(* IEC 61131-3 sources: ml2plc/benchmarks/st (part 4) *)

(* ---- GRU2_straton.st ---- *)
FUNCTION_BLOCK GRU2_FB

    (* Model Inputs/Outputs *)
VAR_INPUT
    input_data : REAL;
END_VAR

VAR_OUTPUT
    output_data : ARRAY[0..2] OF REAL;
END_VAR

VAR
    CONSTANT weights_0_u : ARRAY[0..35] OF REAL := [-1.26034391, 0.836788237, -0.74071312, -1.66741002, -1.1549176, -1.52132487, -1.16551328, -1.43403518, -1.60023963, -1.46855605, -1.58754134, -1.517748, -1.31009662, -0.703322828, -1.11610091, 0.108651124, -1.24668264, -1.7667824, -1.78982019, -1.47540379, -1.49926209, -1.13290668, -1.73071063, -1.48351586, -1.53246319, -2.03121448, -1.50697207, -1.17749131, -1.91584527, -1.08492792, -0.994556248, -1.55253255, -1.03130341, -1.2640295, -0.178557396, -1.63782966];
    CONSTANT recurrent_0_u : ARRAY[0..1295] OF REAL := [-0.0342628956, 0.033126276, 0.0130427806, 0.0238829348, -0.0667412207, -0.0413707495, -0.0313988812, 0.0143869575, 0.190381631, -0.0726102442, 0.0838638023, 0.0527294315, -0.0637015849, -0.182236433, 0.144636199, -0.122772858, -0.141192406, -0.00673655141, 0.0763217956, -0.0320057683, 0.0996292979, -0.137748078, -0.0618084669, -0.0315994285, -0.062908709, -0.00729163829, -0.0906494558, -0.137917697, -0.0289651398, 0.0414582938, -0.0709736273, -0.0059862812, 0.0197576638, -0.0750913471, -0.142621666, -0.0388273448, -0.260161608, 0.00932510011, 0.00876244251, -0.12344873, -0.0972604752, -0.0141034368, 0.07111267, 0.00913770497, 0.170134529, 0.0203112364, -0.0925216526, -0.0673360229, -0.0160743687, 0.117756821, 0.134309813, -0.0970909521, 0.0523982346, -0.0415440686, -0.0711917579, 0.0170196127, -0.045774959, -0.0370751619, -0.0704077557, 0.0188004524, -0.0777330324, 0.283721894, -0.16303502, 0.0651905835, 0.0264630243, 0.0179281905, -0.138563886, 0.0722385198, -0.0791174024, -0.0230214931, -0.163337797, -0.0849895626, 0.00793311652, 0.00964403804, -0.0900170207, -0.0211868752, 0.065747194, 0.141165093, 0.0130933337, -0.126985207, 0.0847581699, -0.195722729, -0.0474834777, -0.0756620616, 0.0745357648, 0.11035046, 0.0613997541, 0.0489263199, 0.0219242349, 0.0518789999, 0.180661157, -0.141433775, -0.0488601774, 0.0343847387, 0.0521875918, -0.0937664136, -0.0139141269, 1.37788593e-05, -0.0523182154, -0.0222289097, 0.199464455, -0.195190653, -0.0105472393, 0.0335475393, 0.17911391, 0.032945402, 0.0335034542, 0.146120399, -0.0346618779, -0.027050646, -0.0628796816, -0.126079142, -0.0608317778, -0.144880667, -0.170438543, -0.139052421, 0.0964757726, -0.0888345987, 0.140413404, -0.00511395978, -0.169440314, -0.0679477602, 0.179598868, 0.0536571033, -0.100946359, 0.297387779, 0.14612335, -0.0515739471, -0.0920707807, 0.1155788, 0.122627199, 0.173509136, -0.0269757025, 0.0626975074, 0.0153822703, -0.128492385, -0.193825796, 0.0969658792, 0.0116878124, 0.0272942241, 0.0452310033, 0.00160261057, 0.264178902, -0.103370436, 0.0297610722, -0.0913388878, -0.0183291547, 0.0166632738, 0.119481407, -0.0304607637, -0.0763635635, -0.000451272033, -0.107587576, -0.151274115, 0.122772105, -0.031456992, -0.000585220521, -0.00406094966, -0.139671892, 0.0299809463, -0.102254301, 0.0713162273, 0.00914381258, -0.0205416568, -0.0607767105, 0.0461449251, -0.0858086646, -0.0383039862, -0.0823218748, 0.0483131632, 0.0267805085, 0.193337917, 0.163598657, 0.0458281264, -0.0303147305, -0.19125393, -0.0151128527, 0.00750773214, 0.0093731042, -0.132128522, -0.0926906914, 0.0911830217, -0.127907664, 0.0237907302, 0.00307789678, 0.0957302004, 0.11556039, 0.172038779, 0.0433095135, -0.0654063001, 0.0514559746, -0.00690185279, 0.0779523849, -0.05985808, -0.135543838, 0.0494517833, 0.0334763303, 0.0388004482, -0.172183558, -0.113222495, -0.142196029, 0.139659673, -0.10881792, 0.0211461224, -0.0613673106, 0.125337034, 0.052437298, 0.0480097719, 0.0614684746, -0.0621075481, 0.215367347, 0.137130678, -0.0973720923, 0.0115704983, 0.254007638, -0.106283039, 0.165332898, 0.173523873, -0.0684746727, 0.0595950186, -0.0305053927, -0.0180566646, 0.0267004631, -0.0547558889, 0.207268775, 0.0180881377, 0.153428495, 0.0346085951, 0.00634628395, -0.0340505242, 0.0254321843, -0.0179827698, -0.110346086, -0.119095467, -0.0225871466, -0.00133527769, 0.115366802, -0.0134922042, -0.130053043, -0.168047309, 0.118532434, 0.16799961, -0.191472441, 0.0312053822, 0.0745509788, -0.0187781006, 0.0191130526, -0.0659152642, 0.113805823, 0.0113544129, 0.178768978, -0.0178589281, -0.173394576, -0.100760654, 0.0929996371, 0.0436356664, -0.0717414394, 0.0160977114, -0.0963451192, 0.195525184, -0.062454652, 0.0209066458, -0.0547173209, -0.0410734601, -0.10283678, -0.00662166253, -0.0165458117, -0.0140010985, -0.0901765451, -0.0117543321, 0.0552607402, 0.0510834008, 0.0607867166, -0.0134733124, 0.0615748167, 0.147052288, 0.120013088, 0.0469233096, 0.0984836742, -0.0120238587, 0.157431439, 0.0271336511, 0.00899497047, 0.0144625632, -0.00717109535, -0.0346801281, -0.0201367103, -0.0010825675, 0.0760441795, -0.0845471472, -0.0586753376, -0.0433512367, 0.0140556972, 0.0254240334, -0.0254383944, -0.00431554019, -0.1569774, -0.0387899987, -0.121743545, 0.229205519, 0.0409585759, 0.0874423534, -0.119842805, -0.0834079385, 0.121145457, 0.0360527039, -0.0465544574, 0.0328435637, -0.039856676, 0.0826937556, 0.0974979177, 0.0160434153, 0.0354771465, 0.216787547, 0.0894127116, 0.0516375378, -0.00532980775, -0.0307577364, 0.0502612591, 0.0561862998, 0.0276951361, -0.00164757669, 0.0275954343, -0.00224959292, -0.0461898521, -0.146057203, -0.0647542998, -0.159321651, 0.0745540559, 0.0591075122, -0.129087731, -0.100868285, -0.0729691386, 0.0610129796, -0.190089911, -0.0530051403, -0.098644577, 0.154064298, 0.0253590234, -0.101725496, -0.0230724476, -0.00965078361, 0.0783198625, -0.0946903601, 0.0650893971, 0.215967342, -0.0486703366, -0.06192315, 0.0585709997, -0.0076801735, 0.18102695, -0.166397452, 0.00742948754, -0.131029949, -0.0124988202, 0.00228013098, -0.0745055452, -0.0188779272, -0.0139701162, 0.066379264, 0.0243779477, 0.173666015, 0.154299214, 0.0105906436, -0.0848416388, -0.192967489, -0.129266128, 0.123107798, 0.0976733416, 0.104287289, -0.126942322, 0.0110000521, 0.107052952, 0.114371777, -0.0595267676, 0.0700232461, 0.068150498, 0.0900249928, 0.0788178518, 0.0185049567, 0.200738877, -0.0606925525, -0.204366297, 0.0851609036, -0.10510283, 0.121970519, 0.0859488249, 0.0492938757, -0.106940009, 0.0186537411, 0.0604228191, -0.163001135, -0.0464588888, -0.00917022303, 0.0485227257, 0.0853310674, -0.159618795, 0.0682769343, -0.0199831873, 0.164003119, 0.193750829, 0.0232146922, -0.100082226, 0.00089744071, 0.216353014, 0.0299245045, -0.00141894538, 0.0168942939, 0.0283064917, 0.00889431499, -0.109997191, -0.0894236043, 0.149576113, 0.0469021723, 0.151476637, -0.120671645, -0.0518624149, 0.102175973, -0.0592916235, 8.79825093e-05, -0.000866604038, -0.153902844, -0.0601970069, 0.180454865, -0.0881382972, 0.0156603139, -0.105296291, 0.0234685838, -0.170900747, 0.194892928, -0.0330442525, 0.15684779, 0.00477843871, -0.235207811, -0.146898672, -0.112256974, -0.0271503665, 0.0876962617, -0.0547677912, 0.000613328419, -0.157910258, 0.111612402, -0.150543317, 0.0749143884, -0.236442089, -0.0640725121, 0.0402319543, -0.129946694, 0.063872084, -0.0921810046, 0.0271176845, 0.0318439715, 0.0775956735, 0.0870574936, -0.177450776, 0.0464093424, -0.033173915, -0.202194497, -0.251605779, -0.0494963601, 0.0495668799, 0.145526662, 0.0401626676, -0.0860805809, -0.0161553323, 0.171846762, 0.0635728985, 0.0118455607, -0.0775468722, 0.0836938843, 0.203875184, 0.000280295033, 0.151499256, 0.00881939288, 0.00597945508, -0.185436562, 0.0678828955, -0.0461877696, 0.0163692199, -0.0452754498, -0.0226855334, -0.0283293016, -0.00942401681, -0.175302401, -0.0285838097, 0.0155983055, -0.0954950303, 0.109856851, 0.035790205, 0.156070665, 0.0800647885, -0.104712404, -0.00879670214, 0.0592416413, 0.0361186527, -0.0642768443, 0.0254080128, 0.0189145245, 0.0923156887, -0.0246102009, 0.0217456631, -0.113064229, -0.0230094828, -0.175723806, -0.0260574259, -0.167376891, -0.0669591501, 0.098559171, -0.0967763886, 0.2555691, 0.0450044125, -0.040658433, -0.0427738503, 0.130444661, -0.0108212894, 0.124109104, 0.00316323247, -0.0725276619, 0.0753806531, 0.112833552, -0.0216558035, 0.0486264825, 0.0383803248, 0.0550877266, 0.00269059022, -0.0247166194, -0.158658102, -0.0149021968, -0.0196858887, -0.0529114418, 0.126081109, -0.0273063388, -0.0963082314, -0.12612091, 0.0636548698, -0.104973838, 0.0937879309, 0.00345468288, -0.13261725, 0.0521132722, -0.0149141084, -0.000320638967, -0.0317318141, -0.0991747305, 0.0467992648, -0.132130101, -0.02635579, -0.034503296, -0.101826586, 0.259196609, -0.0289767701, -0.0308404993, 0.103909321, 0.0277719758, 0.0692727342, -0.184099451, 0.0835822523, -0.030916024, -0.0704697967, -0.135798842, -0.0716379359, -0.153134912, 0.105635196, -0.0149836261, 0.0335508697, -0.0568113029, -0.249705985, 0.0867215171, -0.239200518, -0.0762931556, 0.00669380371, -0.0108323051, 0.213115379, -0.0927517787, 0.0997722, -0.143482327, -0.118950531, -0.0881052837, 0.0756336749, -0.130082756, -0.120683201, 0.02507638, -0.0341131799, 0.0429628938, 0.128947362, -0.124499381, 0.0742484629, 0.168572649, -0.0397992916, 0.00484922156, 0.0362998135, 0.0909697711, 0.0851615295, 0.0326837674, 0.0967172384, -0.164775431, 0.133798763, -0.0326880589, 0.12737225, -0.104726285, -0.0680180341, 0.113625899, -0.0860326439, 0.0464370772, 0.0635163933, -0.0395358279, 0.0639582425, -0.102211565, -0.206772327, -0.00179486861, 0.0213710014, -0.00713133439, 0.086441122, 0.144096032, -0.0194443036, 0.00776778115, 0.104372926, -0.0283569582, -0.0166534446, -0.0287866369, 0.073207587, 0.027669685, 0.0335607752, 0.0479009971, -0.0884077847, 0.0261177346, 0.00300545711, 0.0921291932, -0.0663990453, 0.0354057476, -0.0562885404, 0.0839682892, -0.185307056, -0.0240491442, 0.031400498, -0.173876092, -0.0228056069, 0.106864773, 0.0587361939, 0.0631659254, -0.106001921, 0.0327882767, 0.027667813, -0.000188433682, 0.104556136, 0.252043188, -0.188186049, -0.0209656842, -0.00906039588, 0.0101046152, 0.00515822647, 0.0542920753, -0.0120776091, -0.147997424, -0.00374030834, 0.00196849229, -0.083110109, -0.0612808429, -0.104772605, -0.0237853508, 0.029189622, -0.0479342937, 0.182290047, -0.0171541572, -0.116192788, 0.00495796418, -0.0664217845, 0.000124222715, -0.152234718, 0.0825517401, -0.00798606314, -0.00145258021, -0.0729855448, -0.0400730111, 0.104499131, 0.0208470635, 0.12811248, -0.178114161, -0.0162939616, -0.143496677, -0.10104686, -0.0771575868, -0.108783223, 0.087265186, -0.238202512, 0.0731373429, 0.0663482472, 0.0988706648, -0.0216340423, 0.136428818, 0.0660660267, 0.042084828, 0.157139376, -0.0470077991, -0.112456925, 0.022005707, 0.141990617, -0.0214068051, 0.0737084001, 0.0327303857, -0.0905588195, -0.0811682418, 0.0603267811, 0.0413201973, -0.0958298743, 0.128329098, -0.0242319815, 0.0195612404, 0.0896662176, 0.00108809827, 0.0442191586, -0.188646525, -0.0705579817, -0.0461639129, 0.00824915804, -0.186587214, 0.0156664774, 0.094665125, -0.020454444, 0.0515801646, -0.0784645006, -0.121526279, -0.0748484284, 0.0629792735, -0.0993877351, 0.0471784621, -0.0723702237, -0.158697069, -0.0418656245, -0.0141078103, 0.121266007, -0.123044692, -0.0560409464, 0.00813549757, -0.149031252, 0.0582474172, 0.00461665075, 0.0790261254, 0.194236234, 0.0722888261, 0.0277158916, -0.082633242, -0.136622623, -0.132645652, -0.0448877364, -0.0276510827, -0.144985184, -0.00701641012, -0.0230225436, -0.141255856, 0.144060358, 0.181640565, 0.0743258893, -0.0173662901, 0.111702807, 0.0463593416, 0.035152968, 0.157504857, 0.057882309, -0.032248266, -0.1410629, 0.125498801, 0.037084274, -0.20863165, 0.0922927856, 0.0244627073, -0.17319563, -0.0826953053, 0.0773766935, -0.0771493688, -0.0638951808, -0.128577307, 0.0146199707, 0.0909995288, 0.162200466, 0.00195189286, 0.00804296974, -0.0457642637, 0.0440985113, 0.0135638798, 0.124087267, 0.00408732425, 0.0267615821, 0.0163110215, 0.026695868, 0.00745118596, -0.100966968, -0.0405169912, 0.141835764, -0.0243738946, -0.0111552794, -0.0659039468, 0.149110287, 0.0194932632, -0.0781623721, 0.126755252, 0.0643382519, -0.0551815145, -0.0441562086, 0.00845670514, -0.0503823534, -0.0554201677, 0.000320583582, -0.158687234, -0.170876443, 0.105813354, -0.0343146101, 0.00350035448, 0.00376649201, -0.0166658033, 0.156666756, -0.118631311, -0.0811850652, -0.168449625, -0.1761204, -0.0920138583, 0.0563289449, 0.0803810135, 0.109149583, -0.133163229, -0.134063154, -0.0671341345, 0.0589202866, -0.0166616552, -0.0767766535, -0.0193739664, -0.058711797, -0.198925197, -0.0634987205, -0.0983531401, 0.0787134767, 0.0666048452, 0.045716919, -0.148093581, 0.0425000712, 0.0316398218, -0.0440953895, 0.131269962, -0.0458537526, -0.0241487306, 0.0373034403, 0.00948363543, 0.0806063339, -0.0335490815, 0.0165324025, -0.0595944077, 0.0129592288, -0.0465285331, 0.16187948, 0.179913178, 0.11799854, -0.0625137612, 0.0526206158, 0.0245764926, 0.106756382, -0.121652514, -0.0826648176, 0.010032543, 0.0614630207, -0.00215424201, 0.0180236287, 0.098053515, 0.00795044936, -0.104563564, -0.0765728131, 0.128490895, -0.0422730185, 0.0865375176, -0.170130268, -0.0447101556, -0.126327187, 0.0661132783, 0.0610173345, 0.0859865397, 0.0392063558, -0.0140606016, 0.0137465307, -0.0331719257, 0.00598986261, -0.00775628444, -0.0703896508, -0.0581490695, 0.0697719008, -0.0963044316, 0.0237137936, -0.0178493336, 0.0918230489, -0.0487630256, -0.113788404, -0.188611865, -0.0435639583, 0.0429147929, -0.0721804798, 0.00251296, -0.0345735513, -0.0881643072, -0.0914318636, -0.0498093143, 0.000874343328, -0.0717313141, 0.0340099782, -0.0471353196, -0.0614696257, 0.0318738893, -0.0168175865, -0.0688377097, 0.0278517976, -0.0298618972, 0.0201112907, 0.0501511209, -0.0782770067, -0.0177281275, 0.158253178, -0.108046979, 0.0310336426, 0.0274111014, -0.130947798, 0.0879394263, 0.0393080749, 0.0313053913, 0.0141980154, -0.108860224, 0.0709069371, -0.161655933, -0.160348192, -0.00553186564, 0.13833186, -0.100706764, 0.137516141, -0.137374088, 0.152492315, 0.0974649191, -0.0716144219, 0.280887246, -0.0581361353, -0.0688263699, -0.115718402, -0.0449651927, 0.0464258008, -0.0439850427, 0.145317942, -0.0744717866, -0.199720353, 0.0019946103, 0.0603439175, 0.061749924, 0.118242741, 0.0834349245, 0.0398561172, 0.165977299, -0.0418723375, 0.121971667, -0.077465862, 0.0153007647, 0.0620266907, 0.0509925634, -0.0457279049, 0.158203393, 0.0247548595, -0.0389468186, -0.089520134, -0.170903638, 0.0359030813, 0.0641999766, -0.0221759994, -0.0570958741, 0.0212981645, 0.0752370581, 0.0695017204, -0.0630365908, -0.00289914757, 0.188688084, -0.0300303996, -0.0143778939, 0.0212290064, 0.0268473104, -0.0495267063, -0.023814857, 0.151920021, -0.172052309, 0.0267928932, 0.132540464, 0.0356763862, -0.0396717936, 0.00512547232, 0.0489174463, -0.085691832, 0.00766285416, 0.0522221215, -0.0892943516, 0.124302201, -0.0303064901, -0.218514159, -0.16778478, 0.0532970056, 0.182008982, 0.0896946117, 0.155715063, 0.106090322, -0.0298019443, -0.000262262125, -0.0150951147, -0.159479916, 0.083016336, -0.0419710875, 0.137613669, 0.203732967, 0.0485939272, 0.143195361, 0.126828998, -0.187246934, 0.000569945434, 0.0765563101, 0.110018574, -0.149945021, -0.00629522232, -0.135067254, 0.0676916093, 0.0423727892, 0.0161591545, 0.0520907491, -0.0230580587, -0.0221038107, 0.119314954, -0.0241500996, -0.0610943101, 0.028209962, -0.0757574961, 0.0734885707, 0.0174413025, 0.162281618, 0.155303642, 0.0490410253, 0.075105384, -0.069984071, 0.0564428419, -0.037442144, -0.151975617, -0.194819957, -0.112644881, -0.259342402, 0.0815506279, -0.0968981087, -0.0596687533, -0.00531158503, 0.218267724, -0.00466178637, 0.00406845333, -0.0761522278, 0.0711187273, 0.0261362195, 0.120683044, -0.0166738555, 0.118392497, 0.0102295363, -0.0218743831, 0.0218427889, -0.0687597841, -0.112420656, 0.0128892642, 0.0405472741, 0.0536809154, -0.205715179, -0.178774327, 0.114278913, 0.0123347547, -0.0745173544, 0.201526254, -0.0155321183, -0.024825789, -0.0445906185, -0.0479508601, 0.149425447, 0.0212737583, 0.0346917324, 0.0517859347, 0.0475157648, 0.00832345337, -0.02666042, 0.0999570116, -0.0642044693, 0.0995197073, -0.0150419287, -0.0735240132, 0.0589960255, 0.0344193093, -0.0487776846, -0.0292578507, -0.104162499, -0.0631055236, 0.00468002865, 0.0581661761, -0.173955843, 0.113681093, 0.0185017176, -0.0346038081, -0.128626391, -0.193500057, 0.0346945301, -0.00178579427, 0.00224026339, -0.231290027, 0.245037988, -0.0170679167, -0.0190091208, 0.024668565, 0.0981746763, 0.0367740393, 0.0883608535, 0.0558700152, 0.126212835, 0.0173344314, -0.114995688, -0.176611125, -0.0654156134, -0.0857094601, 0.0865140483, -0.0360516831, -0.0196933392, -0.107615076, -0.0253942609, 0.105702914, 0.0737192109, 0.0108834654, 0.0420503318, 0.00524156215, -0.0134323481, -0.111208729, 0.0618252531, -0.181399539, 0.207519874, 0.0183388703, -0.0395351835, 0.0610462837, 0.143421188, 0.163650081, 0.021800667, 0.0941204131, 0.0145952562, -0.041628439, -0.0158183966, -0.0373831056, -0.0108524635, 0.282158315, 0.0576906241, 0.077838853, -0.0731582567, 0.0125028351, -0.0522309095, -0.13577272, 0.235110492, 0.166962385, -0.0897412151, -0.000142519828, -0.0506511219, 0.09046828, -0.154975027, -0.0405468792, -0.0008863681, -0.126957744, 0.00956340879, 0.0842779353, 0.186090752, -0.123153858, -0.0292314906, -0.0544836298, -0.104556009, -0.0470990986, 0.10033571, 0.130792215, 0.00844831299, -0.0310752168, 0.0321860015, 0.0297145229, 0.1104123, 0.191848353, 0.0397256501, 0.0756020024, -0.0843236148, 0.0389422402, 0.0248937365, -0.0358019099, 0.0566918291, -0.0487754643, -0.0374667458, -0.0647875145, -0.234415397, 0.0179012604, -0.160337508, -0.0247144494, -0.0251942966, 0.168962851, 0.0107776234, -0.0786816031, -0.0342518613, -0.0750932619, 0.079015553, 0.0614081733, -0.122922681, -0.129052252, -0.245205209, 0.0278388374, 0.047563374, 0.0797996968, 0.130940124, 5.15113352e-05, -0.0217881575, 0.1004012, 0.0281585492, 0.170561835, -0.108472809, 0.0389951915, 0.258194625, 0.0529453382, -0.0899566039, 0.175785333, -0.00331248157, -0.108526126, 0.0612452924, 0.157775432, 0.0250135791, 0.110492639, -0.149341404, 0.017977681, -0.0624284931, 0.212826639, -0.077639319, 0.0104098618, -0.00684571452, -0.0996180028, -0.147250965, 0.0354447365, -0.0444453545, 0.233781546, -0.103450991, 0.0155170253, -0.0473377891, -0.0947341919, -0.0377699472, 0.127587453, 0.165696159, -0.136780113, 0.0529446639, 0.165482327, -0.0952069163, 0.0266316608, -0.0179616138, 0.0483686142, 0.0448171496, -0.0421689264, 0.14323771, -0.0839555338, 0.132980764, 0.0211197827, -0.0442603603, -0.050757546, 0.0357376635, -0.125338897, 0.147064731, -0.000512108905, -0.161149159, 0.046065703, -0.117624745, -0.0454183742, 0.145375147, 0.0277413279, -0.0165090188, -0.00931858737, -0.0810929686, 0.0199742056, 0.115814999, -0.0250481963, 0.123653866, -0.0354949906, -0.0402940363, -0.0283595808, 0.14811568, 0.0800062642, 0.00339751877, -0.098010689, 0.0854745582, -0.027271755, 0.0413561799, 0.0582972728, -0.0765109211, -0.0835772753, 0.0691362321, -0.0935782939, 0.109088115, -0.159106135, -0.110543907, -0.0140815703, -0.0383499153, 0.0661629736, 0.128307655, -0.0204003602];
    CONSTANT bias_0_u : ARRAY[0..35] OF REAL := [-3.31684184, -1.92253804, -0.600549936, -3.69921827, -3.10943699, -3.22139859, -3.07832456, -3.3359921, -3.60301566, -3.52053499, -2.0629518, -4.32950211, -3.56971788, -3.00755692, -3.2657485, -3.22026801, -3.31183887, -3.4076972, -2.11697173, -3.42525315, -3.07054067, -3.36058521, -1.97966957, -3.91755629, -3.56717491, -4.29214811, -3.49467325, -3.36011696, -4.08125401, -3.62208104, -2.94322586, -1.91496933, -3.28989291, -3.30953813, -0.811589181, -3.67579985];
    CONSTANT weights_0_r : ARRAY[0..35] OF REAL := [-2.20337677, -1.88937557, 1.01840889, -1.95725238, -2.10569525, -1.84435475, -1.86453593, -2.0972569, -2.23118854, -2.07661414, 1.45937359, -2.47551703, -2.38022447, -2.05377269, -2.04564905, -2.19036245, -1.82878566, -2.17881227, 1.77570093, -2.06604242, -1.720981, -2.00067377, 1.76864231, -2.29959989, -1.94687343, -2.47971582, -2.16341305, -1.92766213, -2.39000511, -1.95265937, -1.64149451, 1.21715331, -1.94317174, -2.12664294, -0.118684582, -1.96202302];
    CONSTANT recurrent_0_r : ARRAY[0..1295] OF REAL := [-0.0518532209, 0.0100792348, 0.0995031521, 0.0562076755, -0.117578536, -0.0814097226, 0.0314493291, 0.098690778, 0.0334832221, -0.202033013, 0.106257744, -0.165642485, -0.127944574, 0.0946999118, 0.0594121329, -0.0588808246, 0.133187503, -0.0501480326, 0.0482184067, 0.102500744, -0.0512330532, 0.100172848, -0.0353195406, 0.0767591149, -0.0616952777, 0.0616215765, -0.072152473, -0.142590791, 0.0253773462, 0.0873886943, 0.0627515018, -0.0060020797, -0.0110717425, -0.11561197, 0.0910828859, 0.0674294531, 0.0674368441, 0.067603305, -0.0291701648, -0.0524768233, -0.153474629, 0.0495595746, -0.0333975703, 0.0105690835, -0.0569075309, -0.123192497, 0.0681755394, 0.056214679, -0.111764096, -0.000123831443, 0.000995786861, -0.0887602046, 0.068499811, -0.0395215191, -0.258146644, 0.00621622242, -0.0951350033, 0.0469855964, -0.113230564, -0.0757883266, 0.133201689, -0.217605323, -0.00608205702, -0.0847553387, -0.0822716281, -0.15144217, -0.0603607632, 0.0511763394, -0.170682341, 0.0520197339, 0.0402875654, 0.0177042149, 0.00151703146, -0.0603645258, 0.041296415, 0.0340809859, 0.100879528, -0.0286527611, 0.131083667, 0.0532704815, -0.141288444, 0.0506049022, 0.131290719, 0.00215459941, -0.0980387479, -0.186562747, -0.0433423743, 0.0188932028, 0.0164522994, -0.047820393, 0.138713464, 0.0501590706, -0.0791536197, -0.095197618, -0.116016597, 0.142612576, -0.0834967643, 0.0732431412, 0.0394586027, 0.0562297665, 0.0174042787, 0.129350141, -0.0260425434, 0.165490314, 0.010483114, 0.141869515, -0.112036049, 0.176090881, -0.1067001, 0.0662041083, -0.0877013654, 0.149817392, 0.173448488, 0.119827077, -0.0273726396, -0.0792291611, -0.0152004361, 0.0514006019, -0.128296986, 0.11975877, -0.0690590069, -0.0972306281, 0.286197215, -0.109886199, -0.0588776432, -0.024349317, -0.0488271303, -0.00500079058, 0.0753225014, 0.0364711694, 0.0682245567, 0.0365205929, -0.282321811, 0.0218460485, -0.089949578, 0.080596, 0.0498538762, 0.0404125936, 0.0352125205, -0.0547977947, 0.0782399103, 0.00291358074, 0.0343199596, 0.0244415328, 0.121812396, -0.0896032304, 0.116393022, 0.106241778, 0.114141345, 0.0388549678, 0.152886912, 0.0611638166, 0.183587626, 0.157235309, -0.0431555398, 0.0564921238, -0.0948063359, 0.182150811, 0.0194190051, -0.0682585686, 0.151916385, 0.0102312472, 0.0863997787, 0.116413504, -0.182932153, -0.0177681744, 0.00379546452, -0.0789515227, -0.15136902, -0.0196578819, -0.191564307, 0.0208359323, 0.124643706, 0.0105623938, 0.2526353, -0.13925533, -0.0359610878, -0.0130393244, 0.0351147056, -0.025538845, 0.0616876855, -0.000872181263, -0.0336071663, 0.0435039215, 0.0909110606, 0.0181540027, -0.214902133, -0.0379557982, -0.0762276128, 0.0481353141, 0.0145603167, -0.140832886, 0.0420654863, 0.171657696, 0.125975475, -0.0903143212, 0.0479161702, 0.0110886358, -0.0732504278, -0.112601191, 0.0547676459, 0.0239557996, -0.00538704544, 0.109696813, -0.0307096038, 0.0124149444, -0.0926457793, -0.00464931689, 0.085125275, 0.00322351209, -0.0455691554, 0.244893432, -0.0680050403, -0.286186844, 0.0240143351, 0.0364020132, -0.0318022184, 0.095760867, -0.22077848, 0.0365609154, 0.121885367, 0.0490611456, -0.039566949, 0.0750380307, -0.104757003, -0.0706891939, 0.226130679, 0.0681866333, 0.136562794, -0.0332673751, 0.133232132, -0.0464696623, 0.14627032, 0.169435084, 0.0817999318, 0.17531547, 0.126671463, -0.0645604953, 0.148341879, -0.0385105647, 0.0922968835, 0.169149756, 0.0486348122, -0.0587215573, -0.011319411, 0.0988983139, 0.157245934, -0.025147818, 0.0725217015, 0.100335777, -0.133685902, 0.127056345, 0.035799861, 0.148788482, 0.0542310886, -0.233383134, -0.0843333825, -0.106023081, 0.0775830522, -0.172619, -0.0575407371, 0.0290057492, -0.0701818764, -0.106069162, 0.120000601, -0.0713435262, 0.167415246, 0.0746002644, 0.0694687292, 0.159994215, -0.0272930935, -0.0163594317, -0.155241951, -0.00117120193, -0.0292222016, -0.0518031158, 0.0270177908, -0.0214920528, 0.047606118, 0.102642633, -0.0973055214, 0.00627216743, 0.0734423846, 0.123990752, -0.0876427516, -0.0488393456, -0.126777112, 0.00610731542, -0.0871917829, 0.163736969, 0.00666533038, -0.0266870297, -0.042937398, 0.0817313492, 0.0953363329, -0.150749162, -0.00827104785, -0.0428364538, 0.122809194, 0.1236367, -0.107383601, 0.114952825, -0.0492989086, 0.0459021479, 0.0617873296, 8.05500313e-05, -0.154523641, 0.265622109, 0.11186444, -0.0223068893, 0.0036137295, -0.0512494706, -0.0734769776, -0.208853647, 0.0959232002, 0.0555404089, -0.0212275963, 0.088280499, -0.100946382, -0.0610488094, -0.0476924181, 0.0427438803, 0.0795567781, -0.0107469689, 0.0199624766, -0.000371331116, 0.229465306, 0.055255305, -0.040757373, -0.20124501, 0.0218797773, -0.113710955, -0.0179725066, -0.0624392629, 0.0917359591, 0.258699626, -0.191937208, 0.0735471994, 0.101364344, -0.00675959513, -0.12078654, 0.0434612371, 0.0274914149, -0.154627591, -0.107847586, 0.00116873847, -0.0447546244, 0.0128801819, 0.0237785038, -0.033341106, -0.0130486619, 0.18131189, -0.109849624, -0.201468989, -0.020951638, 0.0548722669, -0.00318563008, 0.0713363588, 0.0354395136, -0.0785603672, -0.0465192124, 0.123014368, 0.194484815, -0.0414727107, 0.14672339, 0.0671733692, 0.126081288, -0.0929153785, -0.0223649815, -0.052900888, 0.0757329017, -0.0854709968, -0.10499379, -0.0247410443, 0.0331688114, 0.100440755, -0.0271976329, 0.0145992953, -0.030465683, 0.0727633759, 0.00489661191, 0.129947424, 0.0446471237, 0.0272945091, 0.0434387475, -0.118711732, -0.0506779999, -0.211775959, 0.0250467733, 0.0447979011, -0.0494372658, 0.142923221, -0.280163169, 0.0533072874, 0.0044700685, -0.147525981, -0.0704066083, 0.194399327, -0.0774145275, 0.0308785494, 0.0104368431, -0.0486227423, 0.0419197977, -0.000259150635, -0.090705283, -0.0539368242, -0.151456952, 0.0175608173, -0.0166165438, 0.0225642398, 0.037054535, 0.189391986, 0.0128583014, -0.0775838271, -0.0444044992, -0.132277682, -0.0437051281, -0.0157262534, -0.0697432831, -0.29230094, 0.052789893, 0.0444984585, -0.137304708, 0.00351358019, -0.0128398295, 0.0928503722, -0.137720719, -0.0808323249, -0.150143489, -0.111709282, 0.0693309233, 0.0745513886, 0.00160072558, -0.071504429, 0.00779804494, 0.0510330573, 0.0678527728, -0.0809938982, -0.0109598329, -0.0031484433, -0.0168120246, 0.0360189639, 0.0440756008, 0.0447052903, -0.0453105196, 0.199158788, -0.0296272803, 0.0942767784, 0.0714321584, 0.0174807627, -0.0991960838, -0.0637181476, 0.100138254, 0.0168283824, 0.0421470664, 0.0813013762, -0.00397019647, 0.0185558964, -0.0150549505, -0.201667607, -0.0446293093, 0.085110575, 0.0639931038, -0.10885942, 0.121067882, -0.0862203166, 0.0585916229, 0.0124800578, 0.101264425, -0.0807707533, 0.0939626247, -0.123651706, -0.086919412, 0.00486749317, -0.0162009764, 0.0211123191, 0.0556063429, 0.178670168, 0.197959498, 0.0590754487, -0.0808091015, 0.0289960299, 0.110462062, 0.00299698301, -0.0353727043, 0.181408718, -0.0685826018, -0.0113999881, -0.00430076802, -0.0885879844, -0.057933569, 0.0102831693, 0.280484885, 0.0624650046, 0.118355565, 0.0357311554, 0.0632256493, -0.045290567, 0.065026626, -0.147730455, -0.0991021469, -0.027631795, 0.0545543991, 0.113753639, 0.105484247, -0.00100950478, -0.11947988, 0.0837583989, -0.00764888246, -0.022076631, 0.135195524, -0.0310583264, 0.00280306488, 0.146199867, 0.0586315393, -0.0460124984, -0.0389394276, 0.0497984253, -0.125840172, -0.0668842569, -0.10034465, -0.112302519, 0.0681517422, 0.0806426257, 0.256770879, -0.018550884, -0.041362904, 0.0327220634, -0.0266663916, 0.0449167751, -0.0798490942, -0.0270057488, -0.140253633, -0.138583809, -0.108388111, 0.0308570731, -0.109879017, 0.000431412831, 0.0555504858, -0.0449824072, -0.17535682, 0.000755487941, -0.0875047296, 0.0492692962, 0.0203952342, 0.0118262582, 0.0467516109, 0.13168861, -0.0843266547, -0.055955667, 0.0582496636, -0.130700842, -0.141869634, 0.00793353096, 0.0920046419, -0.155876175, -0.00600741617, -0.179789349, -0.115903929, -0.0926623046, -0.0412278473, -0.0603058487, 0.0266902223, -0.143059075, 0.00291747041, 0.129806757, -0.0169999786, -0.163171634, -0.0698610842, 0.00698351394, 0.0591859221, 0.0131016439, -0.00504229125, 0.0735477135, 0.0296590086, 0.0797545612, -0.0487754382, 0.177203476, 0.0872727185, -0.0689574257, 0.187634706, 0.161229327, -0.0239603147, 0.153950647, -0.0511261821, 0.154039338, 0.0571475998, 0.0237450767, -0.230214506, 0.0324941054, -0.0821794048, -0.13773191, -0.054685168, 0.215499967, 0.204144269, -0.115813851, -0.0153602194, -0.0085346112, -0.105144113, -0.078687638, -0.00323357037, 0.0603099652, -0.000601100735, -0.01836868, 0.0746556297, -0.113810159, -0.0355950221, 0.100739501, -0.0066043539, -0.0144560346, -0.00287585799, 0.0465293899, 0.278194815, 0.0537667647, -0.084564127, 0.0477195568, 0.0267558359, -0.15119876, -0.223530829, -0.0112828612, 0.0430232547, -0.0901929736, -0.0839711502, -0.0299314819, -0.0500379428, -0.0052395761, 0.0466068871, 0.00246280991, 0.0858768225, 0.0651532188, -0.0400214903, -0.000787137076, 0.0849189758, 0.0730260611, 0.0207330249, -0.087194182, 0.0584074631, -0.0225706417, -0.0799087957, 0.0632464588, 0.076903373, 0.0482237376, 0.0947350115, -0.0533070713, -0.154844314, 0.00572717283, -0.0188629776, 0.177197486, 0.0635955855, 0.110036597, 0.049848225, 0.0255107973, -0.0921822265, 0.0975539982, -0.0624480359, -0.0511342213, 0.0311849266, -0.0905147642, -0.138580739, 0.0837990642, -0.198811144, -0.109423444, -0.0584463179, 0.127333894, 0.110430174, 0.121374264, 0.010498248, -0.0348857865, 0.202939615, 0.109336242, 0.0188400429, -0.0779666975, -0.0203662626, 0.180037156, -0.00813225657, -0.169715181, 0.0408392511, 0.0624587722, -0.210099861, 0.119841747, 0.0443388373, 0.147961378, -0.0102043403, -0.100028545, 0.214659378, -0.0964728668, 0.112320058, -0.0672991723, -0.035059046, 0.221380159, 0.0784452111, 0.0210489128, 0.105252743, 0.0118561983, 0.0401980355, -0.00723283226, -0.0929713249, 0.168279245, -0.0724994019, 0.0468706638, -0.0974956527, -0.21627976, -0.0665058941, -0.0189923607, 0.064748317, 0.0916003808, 0.146213189, -0.0165754873, -0.00974176452, 0.139920533, 0.0620965809, 0.116363622, 0.0305393487, 0.00690314081, 0.0617128983, 0.153725207, -0.016307557, -0.0443576612, -0.015470406, 0.0893027037, 0.0629043877, 0.105606712, -0.0492847674, -0.0683245659, -0.119380407, 0.0103158439, -0.0134933535, 0.10447222, -0.146812186, 0.0300211795, 0.0904230922, 0.125490665, -0.0684458762, 0.187556997, -0.107997715, -0.0317476168, 0.0650807545, 0.0260817539, 0.20079191, 0.0263294727, -0.123054281, 0.0626507327, 0.142655879, 0.0815112814, -0.0888449922, 0.0381629243, 0.000777062494, 0.0474255085, -0.0742152929, -0.00252578012, 0.0113256313, 0.00749191409, -0.134803012, 0.0964160711, -0.00362235308, -0.00928523019, -0.0167164505, 0.0569139011, 0.051037848, 0.0467544943, -0.0899294242, 0.0371286534, 0.0257632248, 0.0119114388, -0.118839256, 0.0836265087, 0.0157502145, -0.17465122, -0.0546997264, -0.04981016, 0.181788489, -0.0612546727, -0.0582747869, 0.0404811613, -0.0233908743, -0.159590185, 0.0716376156, 0.0204316452, -0.237259611, 0.0772680193, 0.104619272, -0.0421570167, 0.111949079, 0.106285863, 0.107082032, 0.0778088197, 0.270655841, -0.0751747862, -0.0886761472, 0.150075361, -0.0235337317, -0.152854443, -0.0207292326, 0.0644152984, 0.100547396, -0.0542097017, 0.171480745, 0.00509776454, 0.159422144, 0.0197763462, -0.0606458783, 0.0263526067, -0.289731592, -0.120666355, 0.000754584908, 0.0763607025, 0.0298142452, 0.0594509505, -0.0376676396, 0.0499249808, 0.113251172, 0.0301162228, 0.0526147373, -0.133951932, 0.0203451421, 0.151570782, 0.0269404203, 0.0813456401, -0.156112954, 0.0385173932, -0.117552705, -0.123268597, 0.0257833004, -0.0291511379, -0.10322424, -0.0882892534, -0.00362876221, 0.0641316846, 0.00729751633, 0.144065753, -0.0573350303, 0.0278582517, -0.0557212047, 0.0739008933, 0.169447571, -0.070405893, 0.0715222582, 0.115311757, -0.100773193, 0.113157906, -0.186351806, 0.0949108452, 0.0265831146, 0.18958874, 0.0605165549, 0.156304225, 0.0822665021, -0.189060211, 0.143293694, -0.0674860552, -0.0135849854, 0.0239588376, -0.225335628, -0.106712908, 0.0961384624, -0.0832711011, 0.0864122137, 0.208305627, 0.0420468301, 0.0231188796, 0.0580740571, -0.0786098912, -0.0370841101, 0.0332066827, -0.158784777, -0.0544040203, -0.00585781317, -0.180435151, -0.141297638, -0.0778184608, 0.0158938989, -0.0986057594, 0.14170894, 0.131531268, 0.0682063177, 0.0133296726, 0.0215558596, 0.106123649, -0.0551676974, -0.0848584324, -0.019054452, 0.0365033709, -0.0512739532, 0.0370680019, 0.0357793197, -0.103004523, 0.0244357474, -0.0840907246, -0.037492156, 0.0367729552, 0.0874691606, -0.10022606, 0.149992615, 0.021946121, 0.00904138386, 0.0366227999, -0.128580406, 0.0956582874, 0.0371274054, 0.074402079, -0.00108072709, 0.139384255, -0.0619168282, 0.00493702479, 0.0242130961, 0.0357049704, -0.0834867209, 0.158261552, 0.0363248251, 0.0932637975, -0.0754701421, -0.0149764083, 0.064161025, 0.0231743883, -0.107822672, 0.0800110921, -0.0659031197, -0.0165662635, 0.00417651003, 0.124901459, -0.00140193757, 0.0352313034, -0.0714306533, -0.064536795, 0.0669716969, 0.104574569, 0.0706970021, -0.112585515, -0.141672954, 0.0427056924, 0.182428166, 0.0624094643, 0.0167079382, -0.0581905842, -0.0685651526, 0.00562047167, 0.140159935, 0.000948427245, -0.0711839199, 0.13566114, 0.00985746644, -0.222275078, 0.105873942, 0.0330946967, 0.103792652, 0.00625154888, 0.151920617, -0.020965727, 0.0182321928, -0.0968041718, -0.0876097828, -0.0394545496, 0.15104267, -0.157202333, 0.147064045, -0.0732066855, -0.0270045288, -0.0101193544, -0.0686650798, 0.110081613, -0.0291167945, -0.102851212, 0.0635612532, -0.100097306, 0.102936342, 0.0140077248, 0.0113121793, -0.00869001355, 0.05701432, -0.0836130232, 0.0245692655, 0.0396046415, -0.0357317254, -0.174141049, 0.175789908, 0.0577150956, 0.00725003798, 0.211774498, -0.0524472259, 0.145916745, -0.0547990575, 0.0124867884, 0.113892727, -0.116240412, -0.0377078839, 0.0142874215, 0.0772671849, 0.0941549689, 0.215182528, 0.0637049451, -0.046919018, -0.10287194, 0.0552797355, -0.115051053, 0.0198550001, -0.162566021, -0.0283041708, 0.00347376615, 0.0134093612, 0.0667946637, -0.138480082, 0.0428397283, -0.13020727, -0.00962569751, 0.0153936483, 0.0326799713, 0.0314743556, 0.0330662914, -0.0396729633, -0.155417576, -0.183746532, 0.202538714, 0.145398945, -0.0341620147, 0.18969515, -0.144752085, 0.066892162, 0.0863491744, 0.0637069643, -0.0289432872, -0.0746355876, -0.10807281, -0.0594047084, 0.019563375, -0.0975873992, 0.0619184896, -0.158837721, -0.0840504616, -0.0277686305, 0.00164523581, 0.112457387, -0.00887776911, 0.16317451, 0.105846934, -0.00630627386, -0.0486784019, -0.0197759829, 0.0594138503, -0.158485785, 0.00500799529, 0.000954607793, -0.0347631276, 0.12389946, 0.126611412, 0.0285997894, -0.123237364, -0.0927043706, 0.0508534536, 0.138719723, 0.130806863, -0.164398566, -0.0402858667, 0.0704940632, -0.152901039, -0.065903306, 0.145715594, 0.125978574, -0.0462992042, -0.0604482964, -0.181761861, 0.0944116116, 0.0873068944, 0.0544018708, 0.0250987355, -0.0209466983, 0.0193976611, -0.187519148, 0.133329079, 0.0857701302, 0.162598684, 0.0393219776, 0.0143709052, 0.0202042703, 0.130270973, 0.049135793, -0.0385793187, -0.229150653, -0.114346512, 0.0296484418, -0.17166318, -0.0189124569, 0.114376441, -0.0847874507, -0.251479924, 0.130232036, -0.0415646173, 0.0793688968, 0.195719004, -0.058173161, -0.0780674368, -0.0341971777, 0.0277362466, 0.0262693111, 0.0783189386, 0.0322514102, 0.13903749, -0.12970449, -0.0714526922, 0.0993738919, 0.0772460923, 0.078241691, 0.0361125581, -0.0578194894, -0.0525650829, 0.161012843, 0.0176019277, -0.117420316, 0.0452685356, 0.0819206536, -0.124885939, 0.046633292, 0.0662092716, 0.171433896, 0.0437411368, 0.00773426052, 0.025762843, 0.0908774287, 0.104776546, -0.0380901657, -0.0214494616, -0.0406752639, 0.119940892, 0.00902049057, -0.120859176, -0.0927580446, -0.0960092023, 0.0109141385, -0.10416019, -0.0101449434, 0.175696939, -0.0188610293, -0.00950361509, -0.113621809, -0.0160971172, -0.110499717, 0.088303633, -0.0391953848, 0.135602072, -0.133146778, 0.142486155, -0.0670467764, -0.0667726994, -0.0318981558, 0.0184325762, -0.0623606481, 0.121785462, -0.0928524658, -0.0539297312, 0.172238126, 0.143134251, -0.00724053942, 0.0593012348, 0.0201384258, -0.0321100764, -0.203329578, -0.188647941, 0.0070950524, 0.130964041, -0.0529687442, -0.0948252454, 0.199646756, 0.0159571785, 0.0358581692, -0.134549573, 0.143163338, 0.113373071, 0.136311591, -0.0178266186, 0.00802107994, -0.122720428, 0.140263334, 0.0340153687, -0.0322497226, -0.0332209691, 0.0357593521, 0.139840603, -0.0984338596, -0.00311255525, -0.0351548716, -0.161228582, -0.0394239277, -0.00481188763, -0.00701641385, -0.0953010544, -0.0853239298, 0.104423419, -0.105433077, -0.0824452415, 0.0304547604, -0.0574560091, -0.0807900801, -0.0348426104, 0.0112409797, -0.0974811614, 0.079050459, 0.0749837384, 0.035888914, -0.0552931055, -0.0240268521, -0.0802263245, -0.117834389, -0.139057532, -0.0263098739, -0.0357970819, -0.131651193, 0.126278698, -0.118751362, 0.155718952, 0.0594404899, 0.0687793046, 0.0179062579, 0.130389586, -0.170448199, -0.0171591081, 0.0300051272, 0.0431111939, -0.0107906619, -0.098702997, 0.0113696139, 0.033739876, -0.125458106, 0.00529369898, 0.0275769029, -0.0373628214, 0.0516339056, 0.0116728982, -0.0315926969, -0.0585882924, 0.11019817, 0.112982363, -0.219484806, 0.0926488042, 0.241615802, 0.158006221, 0.0785038173, -0.114973284, -0.0791158825, -0.0237597153, 0.0286402795, 0.0847119316, -0.0159554053, -0.0953744948, -0.106541149, -0.0278536137, -0.165073469, -0.0065536215, -0.027385205, 0.00171177159, 0.0896169171, -0.0880253315, -0.00284312479, 0.0144621376, 0.136495546, 0.0131853595, -0.0669229999, 0.0222889688, 0.00116571481, -0.0704545081, -0.0159226842, -0.0797416121, -0.0243039802, -0.00392837543, -0.0344925821, -0.0587737262, 0.0498357713, -0.0683767423, 0.00264115958, -0.0227589831, -0.0755029246, -0.00467891805, 0.00326641556, -0.208050832, 0.0177312046, -0.0274150968, -0.0825206041, -0.0818153918, -0.0801413059, 0.153740391, -0.0957330987, 0.0198270287, 0.195071742, 0.0791128352, -0.0608675741, -0.0716282129, -0.208219916, 0.10542722, 0.0410766602, 0.118620068, -0.197616711, -0.100641593, 0.0202808771, -0.0716520846, -0.023391882, 0.037091881, 0.0524251536, 0.0726265237];
    CONSTANT bias_0_r : ARRAY[0..35] OF REAL := [0.401923776, 0.887989163, 0.580473065, 0.330970556, 0.554839313, 0.233502656, 0.475123644, 0.336207211, 0.420817435, 0.327375829, -0.175557062, 0.652851462, 0.550509691, 0.617028892, 0.552687526, 0.64038223, 0.541880846, 0.488630325, -0.332261652, 0.574186444, 0.19755958, 0.626648664, -0.224227741, 0.622799516, 0.390573889, 0.532325089, 0.550776958, 0.543478668, 0.626356363, 0.695245862, 0.29467997, -0.138495937, 0.567791224, 0.35533464, 0.867575586, 0.352878869];
    CONSTANT weights_0_h : ARRAY[0..35] OF REAL := [-1.67774332, 0.883340597, 0.501028776, -1.65611994, 1.38994503, -1.51615036, -1.51444447, -1.6988523, -1.65848529, 1.65895009, -1.21090555, 1.70891988, -1.84744537, -1.4911319, 1.5453229, -1.34717119, 1.4258914, 1.42102861, -1.49596775, -1.31961942, -1.57374811, -1.54987276, -1.27670288, -1.56382716, 1.52351308, 1.81600785, 1.40919423, 1.61888742, -1.70468426, 1.36580336, -1.52756715, 1.45723128, 1.53714108, -1.59595621, 0.155019373, -1.64721942];
    CONSTANT recurrent_0_h : ARRAY[0..1295] OF REAL := [0.0539476238, 0.159661308, 0.00354639045, 0.0210041329, 0.0331531689, 0.0588548034, 0.0882072523, -0.0643684492, -0.0841050968, -0.111732312, 0.0102705453, 0.0544118956, -0.194359273, -0.0518533476, 0.0809300095, -0.141865239, 0.0777446255, -0.0655298457, 0.230273455, -0.0768015608, 0.0485614501, 0.0840228125, 0.0190300383, -0.0364028178, 0.0786581933, -0.0518973023, 0.104785413, 0.00406502327, -0.0168739315, -0.131169602, 0.0101035014, -0.177550003, -0.00240417453, -0.0610146224, 0.0561776161, 0.0363928042, 0.00483570248, 0.0275399368, -0.0383886173, -0.0370269567, 0.0856645852, 0.0146672195, 0.0961736962, 0.00934588816, 0.145706385, -0.0256946757, -0.0414237864, 0.217776939, -0.00176358409, -0.108390227, -0.0181681458, -0.285528153, 0.0397627503, 0.0077727302, -0.101954579, -0.00588660967, 0.000312425313, -0.116586559, -0.0863923952, 0.0396010913, -0.0358452201, -0.0105776321, -0.0466821902, 0.00958814099, 0.093594268, -0.0966961831, -0.0111363139, 0.0605952591, -0.0668082759, -0.0230648443, -0.112500258, -0.0158293229, -0.0618863404, 0.0462815836, -0.11572744, 0.212124944, -0.174790561, 0.0145971822, -0.0375173092, 0.0692254007, -0.0415483899, -0.0410683081, 0.0437659733, 0.000949346926, 0.0693783611, 0.27178067, 0.218839183, 0.0367260799, -0.0314052887, -0.0207587127, -0.013971894, 0.107745081, -0.0425791889, 0.017705502, -0.0274889544, 0.0160894953, -0.0171394125, 0.0443308018, 0.0132687921, 0.0399717987, 0.0792697966, 0.0211109146, -0.218264595, 0.03772806, -0.0727761909, 0.108575672, 0.0893003792, -0.0592516437, -0.095947884, 0.00859975629, 0.0079933377, -0.0444730073, 0.0514653064, -0.168302238, -0.00851426553, 0.0429772995, 0.137078509, 0.166423008, 0.100148275, 0.0659543574, 0.0986788794, -0.0374533609, 0.0454649478, 0.0380662344, -0.0454511456, -0.108097337, 0.0466935001, -0.0520147495, 0.206409231, 0.217892066, -0.0444457978, -0.0514093861, 0.0516793653, -0.0550018623, 0.0338412635, 0.0303047672, 0.0219713207, -0.0192696452, -0.0157173332, 0.145813197, -0.0389910601, 0.0492426902, 0.0122127589, -0.0370097533, -0.0118557224, -0.149867967, 0.0262359623, 0.185473636, -0.05563391, 0.034003187, -0.0777752995, -0.0177087393, 0.0285816696, 0.0301169064, 0.0943522379, -0.0166731738, 0.0939534381, 0.0842438936, -0.000199469621, 0.071327135, 0.0581350178, -0.0336529985, 0.051483728, -0.0653539971, 0.0634557009, 0.186024234, -0.0368869975, -0.0981858, -0.111612186, -0.0263090171, 0.00747498684, 0.0715175197, -0.142995253, 0.0187128503, -0.0384792127, 0.0493966788, 0.0372526906, -0.048128102, -0.221615002, -0.175192177, -0.0535469092, 0.0821369737, 0.0161486715, 0.0740763992, 0.00328062149, 0.0576167777, 0.0210853592, -0.105628408, 0.0808013603, -0.0685354993, 0.138162091, -0.159240589, 0.057975553, 0.0311315469, -0.016321348, 0.0290355235, -0.0637651235, -0.0154776508, 0.013895724, -0.0797831416, -0.00516906986, 0.0355699472, 0.00791095011, 0.0956009105, 0.0761029869, -0.0966202691, 0.0372279435, 0.0549760982, 0.156587243, -0.243050665, 0.08684019, -0.0908216238, 0.0176242758, -0.0134438723, -0.0398409739, 0.047927916, -0.0411733054, 0.0556228161, -0.109199606, -0.209197536, -0.00440215506, -0.0897763222, 0.024153389, 0.197484434, -0.0646331012, 0.0186560638, 0.0717991143, 0.160821691, 0.0103017185, 0.0642879903, 0.00655157864, -0.116783008, -0.00684507703, 0.165354297, 0.056459073, 0.00215316704, -0.0492985435, 0.0419776626, -0.112154096, -0.0038778903, 0.0847918093, -0.162504479, -0.0272474028, -0.0403930247, 0.0915106535, -0.0176151916, -0.15755637, 0.0279111546, 0.212829202, -0.00299695972, -0.070478037, -0.260667205, -0.105674654, -0.0236216336, 0.0250645764, 0.0592872649, 0.062667869, -0.109310597, 0.0551156364, 0.0490301661, -0.0742225721, -0.0217943955, -0.0177799426, 0.105632812, 0.0444965549, -0.0362950452, -0.0993257165, 0.107500635, 0.0105324993, -0.129555255, -0.0235012621, -0.123549834, -0.141105473, -0.0340937227, 0.00776308356, -0.0043012402, -0.160780445, -0.0510351546, -0.0237176418, -0.00451872963, -0.0295926761, -0.0756147727, 0.0422878489, -0.147121921, -0.148778796, 0.0752051845, 0.0206829682, -0.0289900675, 0.0929051861, -0.00319701782, -0.148432285, -0.0567956492, -0.223374307, 0.0332702436, 0.0363558233, 0.0927929357, 0.0372741744, 0.103176296, -0.0870891362, -0.0294805709, -0.109647721, 0.0184687935, -0.0140496781, 0.00327076763, -0.0530369133, 0.11764238, -0.0481272861, -0.0353967063, -0.143702745, 0.0237285607, -0.035304293, 0.0562506802, -0.0512277521, 0.0403727703, -0.15965645, -0.067994602, -0.116312988, -0.0957446992, -0.0139428861, -0.0463577434, -0.0847203508, 0.0482183509, -0.106707357, 0.153202698, -0.118821599, 0.0385892242, 0.136228174, -0.0789593831, -0.0180123597, 0.116807885, 0.0114439484, -0.0878517479, -0.1810112, -0.0443187691, 0.126365259, 0.0804464519, 0.0793115348, -0.121590443, 0.0120052919, -0.0105328094, 0.0614426844, -0.218111157, 0.109207004, 0.0967407003, -0.0455282331, 0.0874400288, -0.279352814, 0.0668401569, -0.113413468, 0.136496708, 0.0831836089, -0.0272306409, -0.138496891, -0.127923131, -0.128598452, 0.0401502587, 0.0356418528, -0.211472839, -0.0783749297, 0.0507783517, 0.0610476062, 0.0791865811, 0.288531661, 0.0772943869, 0.0516682379, 0.200563401, -0.0272140969, 0.0532903261, 0.0304788686, 0.117516056, -0.0495324098, 0.0709016472, 0.0904448777, -0.0985883623, 0.0152677326, 0.0423569269, 0.0289058276, 0.0801556855, -0.0659915656, -0.0467079729, -0.048654519, 0.105049394, 0.0743180737, 0.188911647, -0.0223209411, 0.0290020145, -0.0823659152, -0.0566085875, -0.0659694523, -0.0956072062, 0.108884886, 0.0527153164, 0.0561773106, 0.0323481373, 0.143082812, -0.167117029, 0.104353271, 0.0289677512, -0.103977524, -0.0224188287, 0.0256763026, -0.025687363, -0.0788785219, -0.0309170764, 0.188142002, 0.0350306891, -0.00972397719, 0.0300678723, -0.104440615, -0.035973914, 0.0201313905, -0.0289865211, 0.12826623, -0.0484686419, -0.133910179, 0.0953613371, 0.0543639883, -0.0841092318, -0.0823651254, -0.0616703294, -0.0788410157, 0.0626801699, 0.304473758, 0.0766542703, -0.0564542599, -0.156051621, -0.0838441774, 0.0927403048, -0.024810357, -0.131124601, -0.0693460405, -0.0393519327, -0.028281128, -0.0384688526, -0.10521996, -0.0926939175, -0.0700246692, 0.185717985, 0.101900801, 0.205355465, 0.0619968139, 0.0712815225, 0.0137632843, -0.201815993, 0.0156218372, 0.0157556292, 0.0546364374, -0.0718404576, 0.154551953, 0.0829650611, -0.019245062, -0.0837980658, -0.0819584429, -0.0340763815, 0.0689055622, -0.190359339, -0.0937107205, -0.131261572, 0.212121338, 0.0952706933, -0.111695133, 0.0535394475, -0.0380665064, 0.109672338, 0.00668391353, -0.0728870556, 0.0478811339, -0.0934191868, 0.021381028, 0.0180425979, -0.0222711749, 0.223898545, 0.101659022, 0.0860073119, -0.0393475443, 0.0295394622, -0.00525387563, -0.0388116799, 0.00481921714, -0.0101829777, 0.0241851918, 0.235109061, 0.0495106429, -0.0115560889, -0.172806919, 0.0890362188, -0.00275856908, 0.147447392, 0.127720699, -0.235859871, -0.0390835702, 0.0980156511, 0.0810236409, -0.114130452, 0.000716209994, 0.0800107569, 0.014007587, -0.0317907259, -0.0372040011, 0.0674476847, 0.0260960795, 0.0708698034, 0.0451841727, -0.256765097, -0.0704066753, 0.0398466289, 0.00720591145, -0.0240614675, 0.132759541, -0.0362602621, 0.183676541, -0.171965197, -0.0605573021, 0.168475404, 0.0729398951, 0.00771710183, 0.068795234, 0.178079948, -0.0210887417, -0.109796681, 0.174324676, 0.109961733, -0.0457612015, 0.0814596042, 0.058647383, 0.0245547313, -0.0674055889, -0.188284963, 0.152298287, -0.0119599197, -0.027047731, -0.0597860627, 0.034427613, -0.00778884254, -0.000835162122, -0.117614105, -0.100326493, 0.027146589, -0.0349072143, 0.000493591418, -0.0226272941, -0.0681159943, 0.060332913, -0.0462313071, 0.0345762521, 0.0430291481, -0.0435643606, 0.153495342, 0.048972968, -0.0736333802, 0.0623482801, 0.0595273487, 0.0621938929, 0.031439323, 0.0615488738, 0.0262554251, -0.176010817, 0.117433921, -0.128584355, -0.00122676615, 0.00980628189, -0.136135295, -0.130859673, 0.0975630134, 0.0119312024, 0.00239557028, -0.10229259, -0.173605323, -0.0170864593, -0.063877821, -0.0646649152, 0.0380217768, -0.027325388, 0.01765671, -0.0497253612, 0.149554104, 0.232655048, 0.0312432796, 0.145675123, -0.130042747, 0.118422866, -0.0170902126, 0.0883590356, 0.0763626546, 0.0576096922, -0.0292969625, 0.152818516, -0.0744025037, 0.0961471274, 0.104938328, 0.0491881333, -0.103883833, 0.120167255, 0.00289875106, 0.011175191, -0.00466636848, -0.0220741853, 0.121481277, -0.136001259, -0.0069872872, -0.19480975, 0.114152305, -0.0559133962, -0.0237097144, 0.0541627407, 0.000819649547, -0.149576947, -0.0734520331, -0.00947207119, 0.152489707, 0.0619721524, -0.0190146156, -0.0202301107, 0.00555088557, -0.134245634, 0.227166668, -0.030286245, -0.0160706341, 0.179680467, 0.0944992453, -0.00310788141, -0.0957225189, -0.00776381046, 0.231903866, 0.0670423955, 0.0515823811, 0.107089221, -0.0889719203, 0.0375059061, 0.216285124, 0.02970252, 0.020662941, -0.0957226828, 0.0884731188, 0.0131082358, -0.0350939706, 0.107688792, -0.0596898831, -0.0150856618, -0.0357639976, -0.0674232244, 0.0086375, -0.0101924632, 0.155443236, -0.0440637246, -0.233757183, -0.059852168, 0.100986414, 0.0308362506, 0.125376523, -0.0679065511, 0.0618300699, -0.0621950328, -0.00278891576, -0.0455510579, -0.128957525, -0.00683484506, -0.0165183824, 0.0323929936, 0.0413387008, 0.0545472726, 0.0122790709, -0.101130925, 0.00489073899, 0.088324815, 0.0783561245, -0.178011417, 0.0228373613, -0.0317489579, 0.0549623966, -0.00934086274, -0.00921998359, -0.0810488686, 0.0626293346, -0.101755977, -0.0806676, -0.0778465793, -0.0647155419, 0.0537022762, -0.0752024129, 0.0580582581, -0.0826500654, -0.00780242216, -0.0150891058, -0.0394765511, -0.122761533, -0.0353822745, 0.00553285424, -0.123092696, 0.0106723085, 0.0571485907, 0.0446273163, 0.10648147, -0.0640488714, -0.127970442, 0.0422729179, 0.0351721421, 0.157700658, -0.205751806, -0.0562551357, -0.182355911, 0.0772750601, 0.00396113936, -0.0887023881, 0.0683497041, 0.0587164536, -0.0566183105, -0.0510265268, -0.0155724939, -0.00545568019, 0.0492211021, -0.120192215, -0.0157710146, -0.160347551, -0.0352062844, -0.0775828883, 0.0439683683, -0.120436855, 0.144028977, 0.0389545858, -0.0797440484, -0.0742567107, -0.0791861415, -0.0475131534, -0.0509591401, 0.00643992517, 0.0578610338, -0.0670297965, 0.033381056, -0.151571825, -0.144670025, -0.0378420912, -0.107657328, 0.0263328254, -0.00296413992, 0.0412168019, 0.247425377, -0.00459840568, -0.122412682, 0.00266740751, 0.102950908, -0.121834733, -0.0280600879, 0.123529531, -0.0238334388, -0.0259227194, 0.128670797, 0.195362583, 0.0875824541, -0.174516931, 0.0254860539, -0.138854295, 0.141168341, 0.0564761721, 0.116196319, -0.103750475, -0.0159229133, -0.151552081, 0.0294401012, -0.0667503625, 0.0561656803, -0.000405230152, 0.0200803485, 0.0305200294, -0.0457499959, 0.11675071, 0.155273482, 0.112394579, -0.0431742333, -0.0864619836, 0.233967528, 0.302560389, 0.15721111, -0.0100201871, -0.0416366681, 0.119899094, 0.126987487, -0.0643069297, -0.054153841, -0.00980899669, 0.0173238702, 0.123024203, -0.100537777, -0.0728107616, 0.045607321, -0.238642767, -0.061329592, -0.134816945, -0.0214728471, -0.085110262, 0.0362270661, -0.0735188872, -0.00869174022, 0.0278634429, 0.0216811839, 0.0642454922, -0.276390105, 0.077331841, -0.097323671, 0.0614526719, -0.029921215, 0.00693411054, 0.0584962107, 0.0170654505, -0.0181061774, -0.0384532586, -0.0454328693, -0.0388103165, 0.0799806714, -0.0395766906, 0.0405838564, -0.0441953652, -0.0941610187, 0.119182266, 0.0830531269, -0.0775224045, 0.0448425598, 0.142063394, -0.104848504, 0.0637661889, 0.175454333, -0.0885748491, -0.0256192572, -0.101015039, 0.146747902, 0.0200363621, -0.128998488, -0.113667682, -0.0690625906, -0.0337796994, -0.151980534, -0.113822021, -0.0291373841, -0.126815647, -0.0921509266, -0.0269419011, 0.104787529, -0.0827619731, -0.077711314, 0.0654826164, -0.0589523613, -0.0493837856, -0.0209197998, 0.0377893224, 0.13397634, -0.140450463, 0.0743217021, 0.171975851, -0.0463676043, 0.00475520547, -0.0419125557, 0.0124535635, -0.0405506715, 0.0149025293, -0.0885443613, -0.0119830072, -0.0391068682, -0.0710843503, 0.161433488, 0.210331932, 0.00608460698, 0.108185209, 0.119318224, -0.10401459, -0.0948734507, 0.0429475866, 0.0217807218, 0.0627988949, 0.00983919576, -0.0651395693, -0.0872698054, -0.158013716, -0.0838020593, 0.0301647708, -0.00434300629, 0.0374769419, -0.0241227597, 0.0910240933, -0.0198380463, 0.114779502, -0.00602585683, 0.0779353008, -0.0662764683, -0.0217418987, -0.0178142153, -0.133407369, -0.0868676901, 0.0122354589, -0.227117851, 0.0525864698, -0.0722999126, 0.0125546511, 0.22632274, -0.0877713934, -0.0218359474, 0.225469768, 0.0475113429, -0.0599466302, -0.0783120692, 0.0350828469, -0.0420980789, -0.0128554767, 0.138522834, -0.0903715268, 0.1247693, -0.0504666008, -0.169042379, -0.0549601503, 0.112816975, -0.25025928, -0.0329325423, -0.000772049418, 0.0273829792, 0.0659241006, 0.0163559858, 0.00552261155, 0.161389917, -0.0451594032, -0.0837665349, -0.140205339, 0.0149619784, -0.233721226, -0.129234031, 0.0921368152, 0.102328472, -0.0737311468, 0.0793932974, -0.0548998639, -0.117187336, 0.103214636, 0.00390645768, -0.0310299955, 0.094068341, 0.118269876, -0.0579105355, 0.167543992, -0.208531901, -0.0147668216, -0.117761195, -0.0961597264, 0.0518684909, -0.101029262, 0.0792476237, -0.0429739654, -0.103600234, 0.0193631705, 0.0641781762, -0.0587958992, 0.00381088629, 0.145095468, -0.0120128039, 0.0828608274, -0.0559775643, 0.059649732, -0.0618158877, -0.104494832, -0.0796408951, 0.122346207, -0.0780295134, 0.0388256274, 0.00900082104, 0.160372734, -0.00298517291, 0.103528246, 0.107281998, 0.193683058, 0.0125377756, -0.147207677, 0.036988277, -0.0181122813, -0.0395720564, -0.0655330941, 0.15920046, -0.128288552, 0.120316215, 0.0575211644, -0.0385373756, -0.000706176739, -0.109130189, -0.156224221, -0.175582737, 0.0836743861, -0.0812146887, -0.0707776845, 0.134519294, -0.0481460132, -0.0187519211, 0.0677945688, 0.0301473457, 0.108377367, 0.00677456614, 0.0823192894, -0.157564715, -0.0393068865, -0.0854738653, -0.164432794, -0.0447419733, -0.0451978445, -0.0869825333, -0.254890919, 0.215797737, 0.0113360928, -0.0285823084, 0.0292423479, -0.0947926715, -0.0100088157, 0.00237392448, -0.0411758162, -0.0553681254, -0.0382645987, 0.146055385, 0.122316375, -0.137937516, -0.132944286, -0.0184058435, 0.110418431, -0.0786418915, -0.0321584605, -0.123529524, -0.0411642455, 0.145534143, -0.00847226288, -0.0227064528, -0.13004297, -0.0118469577, 0.0430590101, 0.128967926, 0.0871081948, 0.0988177657, -0.0993754491, -0.0411155298, -0.121646278, 0.0705653206, 0.0485733785, 0.00625471259, 0.094126381, 0.115968645, 0.0961986631, -0.211373106, 0.0655806065, -0.0747880414, 0.0605820045, 0.126540244, -0.0230597164, 0.105559073, -0.0161375515, 0.0601296462, -0.00640949048, 0.0556308329, -0.129222199, -0.0536417253, 0.0662317723, -0.0780269355, -0.0161563791, -0.0477647558, -0.0487133004, -0.0306010749, -0.0935192853, 0.02975359, -0.141004816, 0.0667223707, -0.0521000065, -0.0842613801, -0.184129879, 0.0497855768, 0.0638667718, 0.157014921, -0.0368853696, -0.0467951931, 0.0771731287, 0.0472973511, -0.0631514192, 0.0904389769, -0.08924485, -0.134929329, 0.079854168, 0.157498762, 0.152604789, -0.0496838689, 0.0659927055, 0.0425110832, 0.129527733, 0.000711719447, 0.114073604, -0.0774358884, -0.0400637649, -0.0568557754, -0.018171126, -0.106267259, 0.0959346965, 0.119391173, -0.0533073358, -0.0529410876, 0.0810947865, 0.195153773, -0.225684702, -0.0612303019, -0.0884686485, 0.00914924126, 0.0438476168, 0.00401067454, 0.0036684128, -0.0950685889, -0.0206606444, -0.158559754, 0.0820208937, 0.129452601, -0.0817669928, 0.0281139612, -0.0478477664, 0.0734263211, -0.023553215, 0.0687638745, 0.00642326847, 0.0840959102, 0.119856052, 0.138040647, -0.0810893103, -0.149980456, -0.0282943211, 0.0953083113, -0.10762018, 0.250854522, 0.0173025709, 0.0502342805, -0.0795894787, -0.0240336601, -0.0663356707, 0.00178683177, -0.033363238, 0.0514662042, 0.204855502, -0.0177310295, -0.0221208986, 0.0908485502, -0.188989937, 0.0199508443, 0.0661074966, -0.169929668, 0.0157565661, -0.020104982, 0.0216266271, 0.060905505, -0.0188193303, 0.0188450478, 0.101562217, -0.0749827325, 0.0187403709, 0.0246638916, -0.125391454, -0.119492233, -0.187690899, 0.0782388598, -0.111457497, 0.0336309224, -0.117860302, -0.0692825392, -0.0635778382, 0.0911167562, -0.0966684148, 0.0381473787, 0.103218116, 0.00540064694, 0.117016353, 0.0219808724, 0.095120348, -0.0804768875, -0.103348568, -0.0555551127, -0.0734853297, 0.0196725037, 0.00230225711, 0.0713690147, 0.109190136, 0.00184574351, 0.0787534043, 0.0162751377, -0.0529042445, 0.0417002887, 0.0513281152, 0.0931230932, 0.10253261, -0.0617204309, -0.00639561471, -0.0178288687, -0.0379109792, -0.204185069, 0.0457139127, -0.0913105384, 0.0141897816, -0.0493329801, -0.0753997862, -0.0210911892, 0.149481893, -0.158560067, -0.223660842, -0.0562594458, 0.106023423, 0.0682478622, 0.156527087, 0.0599901266, -0.101798683, -0.071410723, -0.0267754458, -0.189059258, -0.110498197, -4.21782024e-05, -0.197584018, -0.00378311053, -0.0510116629, -0.179577798, -0.118954197, 0.0198231563, 0.112951957, -0.00869838893, 0.0969041735, -0.0458453223, 0.184820399, 0.0866673365, 0.026595924, -0.0336507373, 0.0167000592, 0.126634881, 0.0161694176, 0.0602932796, -0.0598305464, -0.0428625233, 0.0956569239, 0.0737248883, -0.0264904536, -0.0701940879, -0.00387896644, 0.105184518, 0.168658689, -0.136403382, 0.135669336, -0.0256770812, 0.0769878328, 0.197393, 0.00979706272, -0.0495657399, 0.0257899407, -0.0469679572, -0.0170490034, -0.188964158, 0.0577000454, -0.0488515645, 0.065369688, -0.0322311446, 0.147575155, 0.193704486, 0.00766501017, 0.00449348195, 0.00582372118, -0.153578356, -0.0308619253, 0.0584229417, 0.0790586546, 0.114694752, 0.0263885222, -0.111899152, -0.0275424868, 0.0202123672, -0.0275729112, 0.146062702, -0.0312878527, -0.115136214, 0.0811946541, 0.0845998898, 0.0479431003, -0.00338723417, -0.146811754, -0.225319371, -0.129002944, -0.248497799, -0.0319471061, -0.0981017053, 0.13393952, 0.00314995274, 0.192089632, -0.136918604, -0.0320820212, 0.0309619177, -0.0948490575, -0.0771118999, 0.0492727011, -0.0100245699, -0.00348695088, 0.01345185, 0.009724034, -0.193501279, -0.251503646, 0.0776355639, -0.103028595, -0.0643505529, -0.0250114277];
    CONSTANT bias_w_0_h : ARRAY[0..35] OF REAL := [0.13789767, -0.393039495, 0.230327561, 0.132328033, -0.213968888, 0.0860213861, 0.206931338, 0.10634727, 0.142884776, -0.106363826, -0.00728841964, -0.233300716, 0.219627813, 0.272904098, -0.238475174, 0.289048791, -0.249711528, -0.177586362, 0.0763061196, 0.234076917, 0.101010993, 0.256234825, 0.0102742994, 0.232671976, -0.15997605, -0.182791293, -0.210118607, -0.237912625, 0.254507393, -0.268791139, 0.122710682, -0.00801999494, -0.264012665, 0.115960635, -0.303606927, 0.145280004];
    CONSTANT bias_r_0_h : ARRAY[0..35] OF REAL := [0.572393715, -0.658964396, 0.267485023, 0.423500717, -0.606753647, 0.310276449, 0.444967717, 0.485038847, 0.60597384, -0.470761806, -0.119375296, -0.632520914, 0.739814401, 0.630673468, -0.587485492, 0.70688802, -0.507558465, -0.615021467, -0.135799587, 0.626880884, 0.262894392, 0.52347368, -0.167219713, 0.620650172, -0.446221471, -0.676750243, -0.642188072, -0.485802352, 0.738594651, -0.508656144, 0.306088269, 0.0788854957, -0.575169861, 0.506910205, -0.324196517, 0.434057415];
    CONSTANT weights_4 : ARRAY[0..107] OF REAL := [2.23373985, -0.754756391, -2.03209519, -0.470918506, -0.263014197, 1.37292433, -0.589997232, 0.801350713, -0.180364817, 2.39219809, -0.847354174, -1.82542908, -1.94790435, -0.306766808, 2.3302176, 2.18361425, -0.546861827, -1.25050712, 2.05239677, -0.280096918, -2.16199994, 2.03919029, -0.964660108, -1.73599923, 2.60618234, -0.334174365, -1.91519749, -2.33910108, 0.893779278, 1.74458885, 1.51265132, -0.965512872, -1.04512405, -2.0465343, 0.177311778, 3.05256104, 2.0868814, 0.199072167, -1.87338448, 1.62895453, 0.39870134, -2.16460228, -1.78936565, -0.10534814, 2.33570766, 1.14153075, 0.258192539, -2.13339972, -1.96188509, -0.213608354, 2.50420928, -2.21707582, -0.0259403624, 2.68682909, 1.0372504, -0.698500037, -0.907171369, 1.85397863, 0.46684289, -2.41311908, 1.82555962, -0.680127144, -1.27095342, 1.63660848, 0.128643692, -2.13348198, 1.55462956, -0.688774824, -0.803204656, 1.86154211, 0.089972958, -2.63801551, -2.66718268, 0.606494427, 2.27520132, -2.62292051, 0.602961004, 2.96978164, -1.98853087, -0.299116492, 2.51787686, -1.93966937, 0.0860323533, 2.1084199, 1.90302193, 0.302508622, -2.73465133, -1.25223839, -0.174008667, 2.27427506, 2.25403023, -0.984678388, -1.80594003, -1.32676148, 0.577955365, 0.589322209, -1.89480019, -0.376683116, 2.16545534, 2.46424341, -0.82388252, -1.94319737, -0.0579185821, -0.576541007, 0.723118424, 2.32531428, -0.95584476, -2.07559204];
    CONSTANT bias_4 : ARRAY[0..2] OF REAL := [-0.0344128571, 0.232081696, -0.371323168];
END_VAR

VAR
    (* Merged variables from all regions *)
    buffer_0 : ARRAY[0..35] OF REAL;
    buffer_1 : ARRAY[0..35] OF REAL;
    h_new_0 : ARRAY[0..35] OF REAL;
    h_state_0 : ARRAY[0..35] OF REAL;
    r_gate_0 : ARRAY[0..35] OF REAL;
    u_gate_0 : ARRAY[0..35] OF REAL;

    (* Temporary computation variables *)
    i : DINT;
    j : DINT;
    t : DINT;
    sum : REAL;
    (* Computation helpers *)
    max_val : REAL;
    exp_val : REAL;
    exp_sum : REAL;
    (* Spatial loop variables *)
    oc : DINT;
    oh : DINT;
    ow : DINT;
    ic : DINT;
    kh : DINT;
    kw : DINT;
    ih : DINT;
    iw : DINT;
END_VAR

(* Forward pass execution *)

(* Region: r0 [ACYCLIC] *)
(* Acyclic Region r0 *)
(* Layer 0: GRU (hidden_size=36, input_size=1, seq_len=1) *)
(* Generating output: Y, linear_before_reset=1 *)

(* Initialize states to zero *)
FOR j := 0 TO 35 DO
    h_state_0[j] := 0.0;
END_FOR;

(* Process 1 timesteps *)
FOR t := 0 TO 0 DO

    (* Reset Gate *)
    FOR j := 0 TO 35 DO
        sum := 0.0;
        FOR i := 0 TO 0 DO
            sum := sum + input_data * weights_0_r[j * 1 + i] ;
        END_FOR;
        FOR i := 0 TO 35 DO
            sum := sum + h_state_0[i] * recurrent_0_r[j * 36 + i] ;
        END_FOR;
    sum := sum + bias_0_r[j];
    r_gate_0[j] := 1.0 / (1.0 + EXP(-sum));
    END_FOR;

    (* Update Gate *)
    FOR j := 0 TO 35 DO
        sum := 0.0;
        FOR i := 0 TO 0 DO
            sum := sum + input_data * weights_0_u[j * 1 + i] ;
        END_FOR;
        FOR i := 0 TO 35 DO
            sum := sum + h_state_0[i] * recurrent_0_u[j * 36 + i] ;
        END_FOR;
    sum := sum + bias_0_u[j];
    u_gate_0[j] := 1.0 / (1.0 + EXP(-sum));
    END_FOR;

    (* Candidate (lbr=1): h'_t = tanh(Wx + r_t * (Rh + Rb_h) + Wb_h) *)
    FOR j := 0 TO 35 DO
        sum := 0.0;
        FOR i := 0 TO 0 DO
            sum := sum + input_data * weights_0_h[j * 1 + i] ;
        END_FOR;
        exp_val := 0.0;
        FOR i := 0 TO 35 DO
            exp_val := exp_val + h_state_0[i] * recurrent_0_h[j * 36 + i] ;
        END_FOR;
        sum := sum + r_gate_0[j] * (exp_val + bias_r_0_h[j]);
        sum := sum + bias_w_0_h[j];
    exp_val := EXP(2.0 * sum);
    h_new_0[j] := (exp_val - 1.0) / (exp_val + 1.0);
    END_FOR;

    (* Hidden state: h_t = u_t * h_{t-1} + (1 - u_t) * h'_t *)
    FOR j := 0 TO 35 DO
        h_state_0[j] := u_gate_0[j] * h_state_0[j] + (1.0 - u_gate_0[j]) * h_new_0[j];
    END_FOR;

    (* Y output: Full sequence *)
    FOR j := 0 TO 35 DO
        buffer_0[t * 36 + j] := h_state_0[j];
    END_FOR;
END_FOR;

(* Layer 1: Squeeze *)
FOR i := 0 TO 35 DO
    buffer_1[i] := buffer_0[i];
END_FOR;

(* Layer 2: Slice starts=[0] ends=[1] axes=[0] steps=[1] *)
FOR i := 0 TO 35 DO
    buffer_0[i] := buffer_1[i];
END_FOR;

(* Layer 3: Squeeze *)
FOR i := 0 TO 35 DO
    buffer_1[i] := buffer_0[i];
END_FOR;

(* Layer 4: Fused Linear + SOFTMAX *)
FOR j := 0 TO 2 DO
    sum := 0.0;
    FOR i := 0 TO 35 DO
        sum := sum + buffer_1[i] * weights_4[i * 3 + j];
    END_FOR;
output_data[j] := sum + bias_4[j];
END_FOR;

(* Softmax: find max *)
max_val := output_data[0];
FOR i := 1 TO 2 DO
    IF output_data[i] > max_val THEN
        max_val := output_data[i];
    END_IF;
END_FOR;

(* Softmax: compute exponentials and sum *)
exp_sum := 0.0;
FOR i := 0 TO 2 DO
    output_data[i] := EXP(output_data[i] - max_val);
    exp_sum := exp_sum + output_data[i];
END_FOR;

(* Softmax: normalize *)
FOR i := 0 TO 2 DO
    output_data[i] := output_data[i] / exp_sum;
END_FOR;

END_FUNCTION_BLOCK
